{attribute 'GeneratedUsingTerminal: EL2522-0000-0017'}
{attribute addProperty BoxType "EL2522-0000-0017"}
{attribute addProperty Id "StatusAT %I*Status_70E023F86Counter_valueAT %I*UDINT4"}
{attribute addProperty CRC "2837785672"}
{attribute addProperty Size "10"}
TYPE ENC_Status_Channel_A9252C48 EXTENDS InputBase_8311D824 :
STRUCT
	{attribute addProperty Name "Status"}
	Status AT %I* : Status_70E023F8;
	{attribute addProperty Name "Counter_value"}
	Counter_value AT %I* : UDINT;
END_STRUCT
END_TYPE

(* stored: Version 1.2.0.0, ProductVersion 3.1.4024.11
   DUT ENC_Status_Channel_A9252C48: Id {920942a0-69bc-42e9-8240-d4d1ffe5edff} *)
